# EPICS substitutions: iocs/MC04/MCApp/Db/SAI_DigitalChannels.substitutions
file /opt/epics/modules/SAI/db/SAI_DigitalChannels.template {
pattern {	P,		R,		SCAN, 		ASYNPORT}
        { 	"XF:06BMA-OP",		"{MC:04}",	"1 second",	"pmac"}
}

#EOF
